TYPE ST_TouchProbeGet :
STRUCT
  State           : UINT;   // 0 := deactivated, 100 := BUSY, 1000 := DONE, 9000 := ERROR
  LatchPositive   : LREAL;  // rising edge
  LatchNegative   : LREAL;  // falling edge
END_STRUCT
END_TYPE

(* stored: Version 1.1.0.1, ProductVersion 3.1.4024.12
   DUT ST_TouchProbeGet: Id {53561cfa-a685-44fd-ad0e-5f97b7829672} *)
